Staubli VAL3: getSize.pgx

public program getSize(num& x_nSize[])
begin
  // get the size for the counter
  x_nSize=size(saveInOut:cCount)
  // get the size for the aCounter
  x_nSize=x_nSize+size(saveInOut:aCount)
end
